PROGRAM Heartbeat
VAR
	start_TON: TON;
	start_TON_et : TIME;
	reset_TON : TON;
	reset_TON_et : TIME;
	screen_refresh_pulse : BOOL;
	
	pulse_ms_TON : TON;
	pulse_ms_et : TIME;
	reset_ms_TON : TON;
	reset_ms_TON_et : TIME;
	pulse_ms : BOOL;
END_VAR

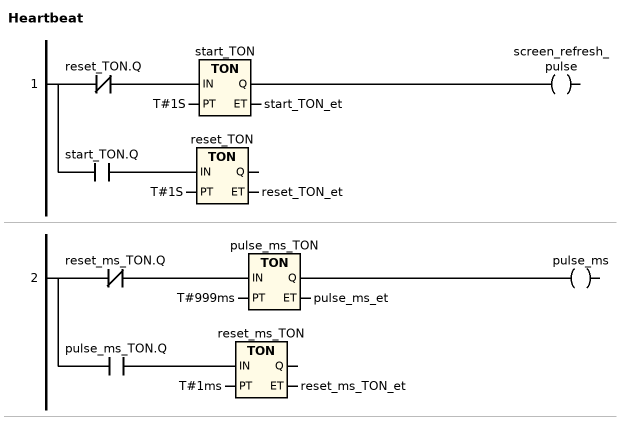
// NETWORK 1
start_TON(IN := NOT reset_TON.Q, PT := T#1S, ET => start_TON_et); // TON
screen_refresh_pulse := start_TON.Q;
reset_TON(IN := start_TON.Q, PT := T#1S, ET => reset_TON_et); // TON

// NETWORK 2
pulse_ms_TON(IN := NOT reset_ms_TON.Q, PT := T#999ms, ET => pulse_ms_et); // TON
pulse_ms := pulse_ms_TON.Q;
reset_ms_TON(IN := pulse_ms_TON.Q, PT := T#1ms, ET => reset_ms_TON_et); // TON

END_PROGRAM

(* stored: Version 1.1.0.1, ProductVersion 3.1.4024.9
   POU Heartbeat: Id {75f70c7f-6977-4f63-8075-a15f4b871ef8}, SpecialFunc None *)
